% RSLogix 500 project SENSORCALIBRATION_BAK004.RSS, saved by version 8.30.00.16 %
PROJECT "UNTITLED"    % processor: Bul.1763 MicroLogix 1100 Series B %

PROGRAM FILES
  LAD 2   3 rungs
  LAD 3 "I/O"  4 rungs  % Inputs & Outputs %
  LAD 4 "CONTROLS"  16 rungs  % Control Logic %

DATA FILES
  O0 OUTPUT  4 elements
  I1 INPUT  6 elements
  S2 STATUS  66 elements
  B3 BINARY  2 elements
  T4 TIMER  2 elements
  C5 COUNTER  1 elements
  R6 CONTROL  1 elements
  N7 INTEGER  15 elements
  F8 FLOAT  1 elements
  L9 LONG  1 elements

LADDER 2
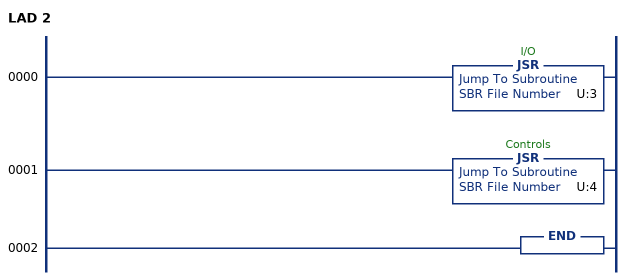
% Rung: 0 %
SOR JSR U:3 EOR
%   U:3  "I/O" %
% Rung: 1 %
SOR JSR U:4 EOR
%   U:4  "Controls" %
% Rung: 2 %
SOR END EOR

LADDER 3 "I/O"    % Inputs & Outputs %
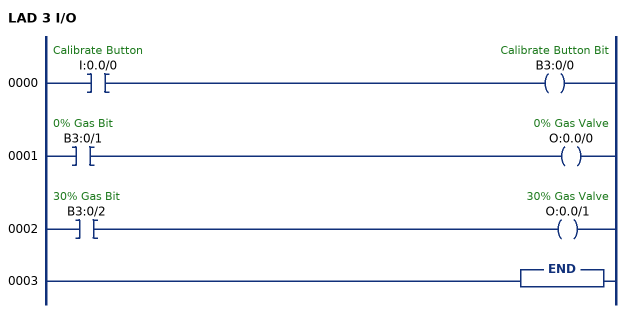
% Rung: 0 %
SOR XIC I:0.0/0 OTE B3:0/0 EOR
%   I:0.0/0  "Calibrate Button" %
%   B3:0/0  "Calibrate Button Bit" %
% Rung: 1 %
SOR XIC B3:0/1 OTE O:0.0/0 EOR
%   B3:0/1  "0% Gas Bit" %
%   O:0.0/0  "0% Gas Valve" %
% Rung: 2 %
SOR XIC B3:0/2 OTE O:0.0/1 EOR
%   B3:0/2  "30% Gas Bit" %
%   O:0.0/1  "30% Gas Valve" %
% Rung: 3 %
SOR END EOR

LADDER 4 "CONTROLS"    % Control Logic %
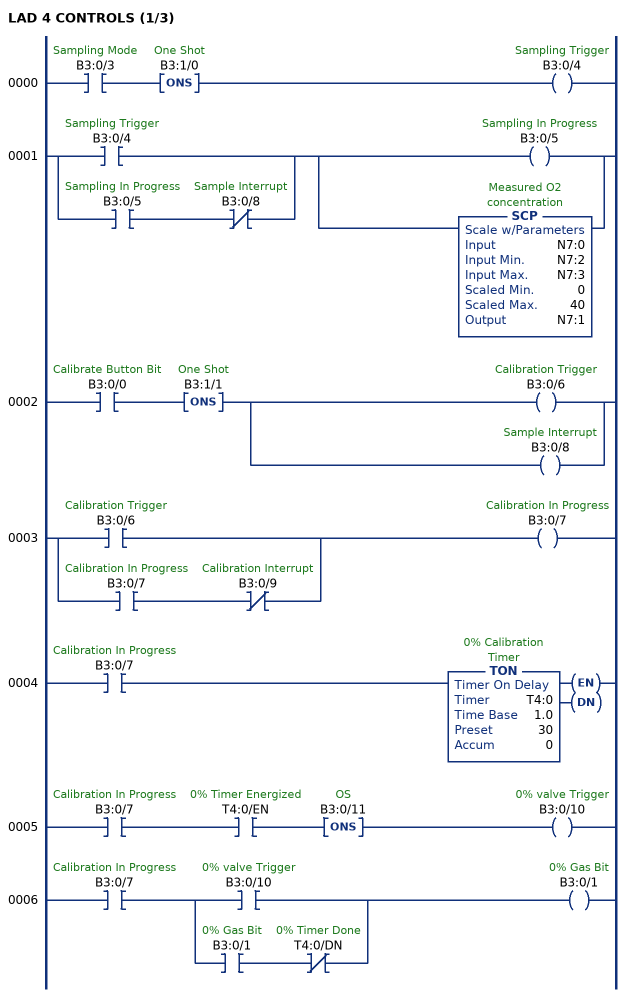
% Rung: 0 %
SOR XIC B3:0/3 ONS B3:1/0 OTE B3:0/4 EOR
%   B3:0/3  "Sampling Mode" %
%   B3:1/0  "One Shot" %
%   B3:0/4  "Sampling Trigger" %
% Rung: 1 %
SOR BST XIC B3:0/4 NXB XIC B3:0/5 XIO B3:0/8 BND BST OTE B3:0/5 NXB SCP N7:0 N7:2 N7:3 0 40 N7:1 BND EOR
%   B3:0/4  "Sampling Trigger" %
%   B3:0/5  "Sampling In Progress" %
%   B3:0/8  "Sample Interrupt" %
%   N7:0  "O2 Sensor" %
%   N7:2  "Calibrated O2 min" %
%   N7:3  "Calibrated O2 max" %
%   N7:1  "Measured O2 concentration" %
% Rung: 2 %
SOR XIC B3:0/0 ONS B3:1/1 BST OTE B3:0/6 NXB OTE B3:0/8 BND EOR
%   B3:0/0  "Calibrate Button Bit" %
%   B3:1/1  "One Shot" %
%   B3:0/6  "Calibration Trigger" %
%   B3:0/8  "Sample Interrupt" %
% Rung: 3 %
SOR BST XIC B3:0/6 NXB XIC B3:0/7 XIO B3:0/9 BND OTE B3:0/7 EOR
%   B3:0/6  "Calibration Trigger" %
%   B3:0/7  "Calibration In Progress" %
%   B3:0/9  "Calibration Interrupt" %
% Rung: 4 %
SOR XIC B3:0/7 TON T4:0 1.0 30 0 EOR
%   B3:0/7  "Calibration In Progress" %
%   T4:0  "0% Calibration Timer" %
% Rung: 5 %
SOR XIC B3:0/7 XIC T4:0/EN ONS B3:0/11 OTE B3:0/10 EOR
%   B3:0/7  "Calibration In Progress" %
%   T4:0/EN  "0% Timer Energized" %
%   B3:0/11  "OS" %
%   B3:0/10  "0% valve Trigger" %
% Rung: 6 %
SOR XIC B3:0/7 BST XIC B3:0/10 NXB XIC B3:0/1 XIO T4:0/DN BND OTE B3:0/1 EOR
%   B3:0/7  "Calibration In Progress" %
%   B3:0/10  "0% valve Trigger" %
%   B3:0/1  "0% Gas Bit" %
%   T4:0/DN  "0% Timer Done" %

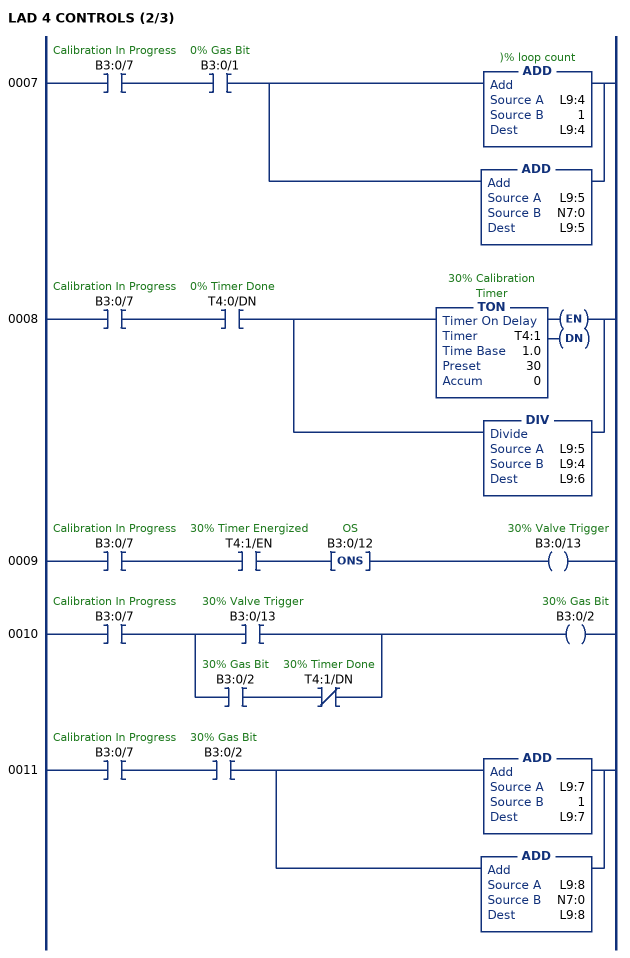
% Rung: 7 %  % edit flag set %
SOR XIC B3:0/7 XIC B3:0/1 BST ADD L9:4 1 L9:4 NXB ADD L9:5 N7:0 L9:5 BND EOR
%   B3:0/7  "Calibration In Progress" %
%   B3:0/1  "0% Gas Bit" %
%   L9:4  ")% loop count" %
%   N7:0  "O2 Sensor" %
% Rung: 8 %  % edit flag set %
SOR XIC B3:0/7 XIC T4:0/DN BST TON T4:1 1.0 30 0 NXB DIV L9:5 L9:4 L9:6 BND EOR
%   B3:0/7  "Calibration In Progress" %
%   T4:0/DN  "0% Timer Done" %
%   T4:1  "30% Calibration Timer" %
%   L9:4  ")% loop count" %
% Rung: 9 %
SOR XIC B3:0/7 XIC T4:1/EN ONS B3:0/12 OTE B3:0/13 EOR
%   B3:0/7  "Calibration In Progress" %
%   T4:1/EN  "30% Timer Energized" %
%   B3:0/12  "OS" %
%   B3:0/13  "30% Valve Trigger" %
% Rung: 10 %
SOR XIC B3:0/7 BST XIC B3:0/13 NXB XIC B3:0/2 XIO T4:1/DN BND OTE B3:0/2 EOR
%   B3:0/7  "Calibration In Progress" %
%   B3:0/13  "30% Valve Trigger" %
%   B3:0/2  "30% Gas Bit" %
%   T4:1/DN  "30% Timer Done" %
% Rung: 11 %  % edit flag set %
SOR XIC B3:0/7 XIC B3:0/2 BST ADD L9:7 1 L9:7 NXB ADD L9:8 N7:0 L9:8 BND EOR
%   B3:0/7  "Calibration In Progress" %
%   B3:0/2  "30% Gas Bit" %
%   N7:0  "O2 Sensor" %

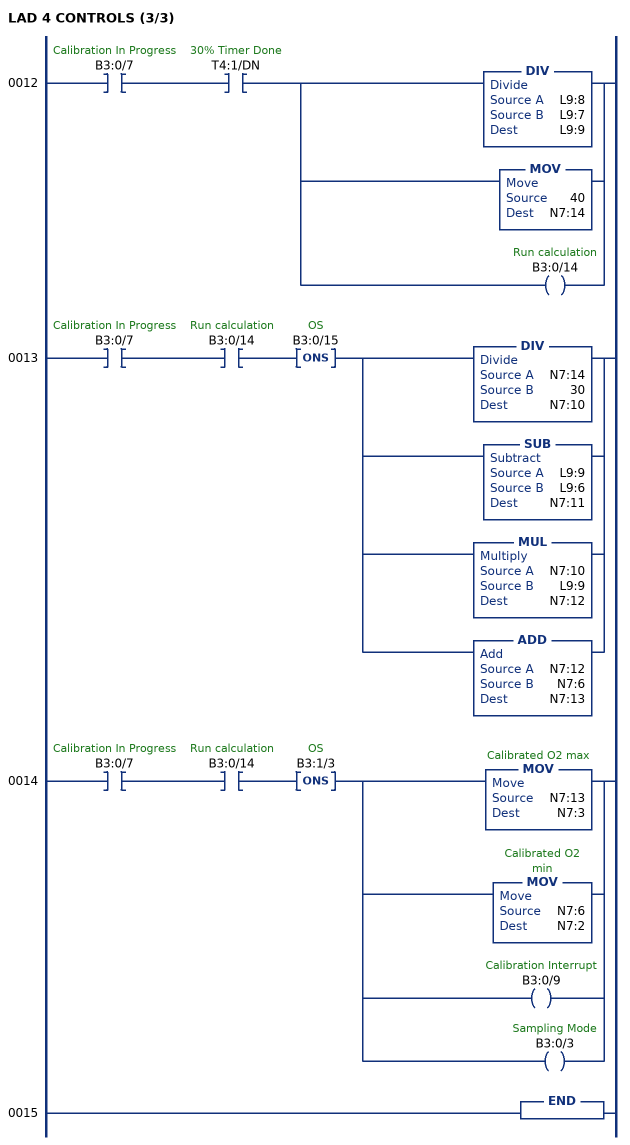
% Rung: 12 %  % edit flag set %
SOR XIC B3:0/7 XIC T4:1/DN BST DIV L9:8 L9:7 L9:9 NXB BST MOV 40 N7:14 NXB OTE B3:0/14 BND BND EOR
%   B3:0/7  "Calibration In Progress" %
%   T4:1/DN  "30% Timer Done" %
%   B3:0/14  "Run calculation" %
% Rung: 13 %  % edit flag set %
SOR XIC B3:0/7 XIC B3:0/14 ONS B3:0/15 BST DIV N7:14 30 N7:10 NXB BST SUB L9:9 L9:6 N7:11 NXB BST MUL N7:10 L9:9 N7:12 NXB ADD N7:12 N7:6 N7:13 BND BND BND EOR
%   B3:0/7  "Calibration In Progress" %
%   B3:0/14  "Run calculation" %
%   B3:0/15  "OS" %
%   N7:6  "0& calibration value" %
% Rung: 14 %
SOR XIC B3:0/7 XIC B3:0/14 ONS B3:1/3 BST MOV N7:13 N7:3 NXB BST MOV N7:6 N7:2 NXB BST OTE B3:0/9 NXB OTE B3:0/3 BND BND BND EOR
%   B3:0/7  "Calibration In Progress" %
%   B3:0/14  "Run calculation" %
%   B3:1/3  "OS" %
%   N7:3  "Calibrated O2 max" %
%   N7:6  "0& calibration value" %
%   N7:2  "Calibrated O2 min" %
%   B3:0/9  "Calibration Interrupt" %
%   B3:0/3  "Sampling Mode" %
% Rung: 15 %
SOR END EOR

OTHER DOCUMENTED ADDRESSES
  B3:1/2  "One Shot"
  N7:4  "0% loop count"
  N7:7  "30% loop count"
  N7:9  "30% calibration value"

DATA TABLE (non-zero values as saved)
DATA T4
% .PRE .ACC %
% T4:0 % 30 0
% T4:1 % 30 0
